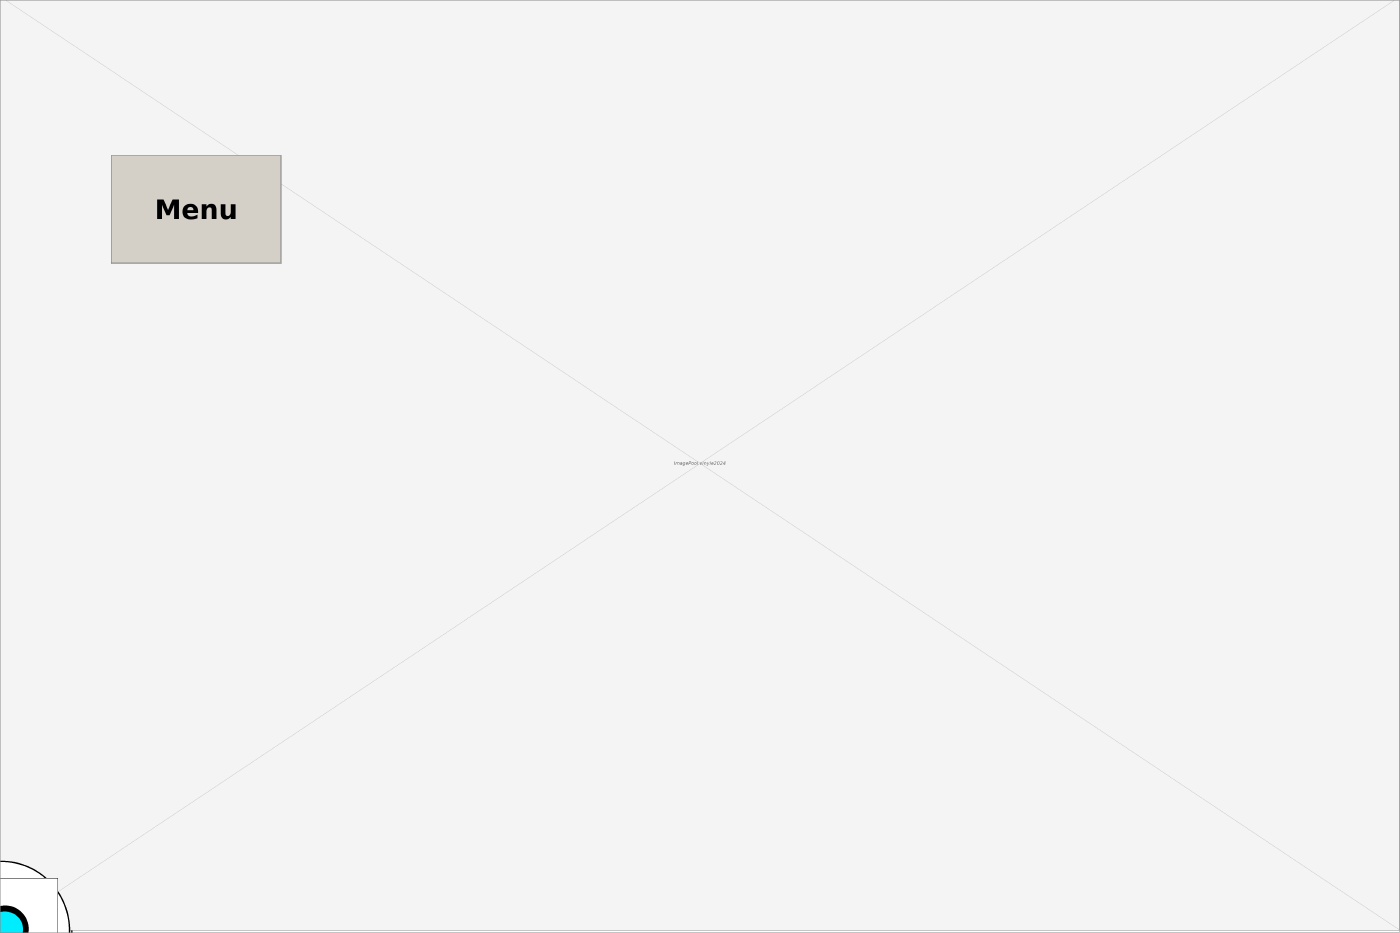
VISUALIZATION V_Deplacement  // 3000x2000
    Ellipse (-142,1844 294x300), "Méchant 1", invisible if: ITInterruption.balise.Nothing1
        p3560616238: ITInterruption.balise.CoordX1
        p2738717112: ITInterruption.balise.CoordY1
    Ellipse (-139,1841 294x300), "Méchant 3", invisible if: ITInterruption.balise.Nothing3
        p3560616238: ITInterruption.balise.CoordX3
        p2738717112: ITInterruption.balise.CoordY3
    Image (0,-8 3000x2002), image: ImagePool.vinyle2024
    Ellipse (-144,1845 294x300), "Méchant 2", invisible if: ITInterruption.balise.Nothing2
        p3560616238: ITInterruption.balise.CoordX2
        p2738717112: ITInterruption.balise.CoordY2
    RoundedRectangle (-102,1882 226x226)
        p2858320360: 360-G_Odometrie.lrAngleDeg
        p3560616238: G_Odometrie.lrPositionX
        p2738717112: -G_Odometrie.lrPositionY
    Ellipse (-39,1941 100x100)
        p3560616238: G_Odometrie.lrPositionX
        p2738717112: -G_Odometrie.lrPositionY
        p2858320360: 360-G_Odometrie.lrAngleDeg
    Ellipse (-74,2050 35x35)
        p3560616238: G_Odometrie.lrPositionX
        p2738717112: -G_Odometrie.lrPositionY
        p2858320360: 360-G_Odometrie.lrAngleDeg
    Button (238,333 365x232), "Menu"
        OnMouseDown: change screen: V_Menu
    Ellipse (-30,1953 80x78)
        p3560616238: ITMotion.odometrie.lrExpectedX
        p2738717112: -ITMotion.odometrie.lrExpectedY
END_VISUALIZATION

(* stored: Version 1.1.0.1, ProductVersion 3.1.4024.12
   Visu V_Deplacement: Id {579fb7f8-a04f-4735-a622-235f82292a92} *)
